(* PLC project Unnamed, Unknown Unnamed 1 *)
(* stored: creationDateTime 2024-09-03T16:04:08, modificationDateTime 2024-09-10T11:48:46 *)

PROGRAM irrigation_LD
  VAR
    SoilMoisture AT %IW0.0 : INT;  (* Soil moisture input from Modbus *)
  END_VAR
  VAR
    SoilMoistureMaxValue0 : INT := 500;  (* Soil moisture upper bound *)
  END_VAR
  VAR
    Temperature AT %IW0.1 : INT;  (* Temperature input from Modbus *)
    Humidity AT %IW0.2 : INT;  (* Humidity input from Modbus *)
    WaterFlow AT %IW0.3 : INT;  (* Water flow input from Modbus *)
    Pressure AT %QX0.4 : INT;  (* Pressure input from Modbus *)
    PumpControl AT %QX0.0 : BOOL;  (* Output to control the pump *)
    ValveControl AT %QX0.1 : BOOL;  (* Output to control the valve *)
  END_VAR
  VAR  (* added by the conversion: wires and edge detectors of the diagram *)
    _LE8_OUT : BOOL;
  END_VAR

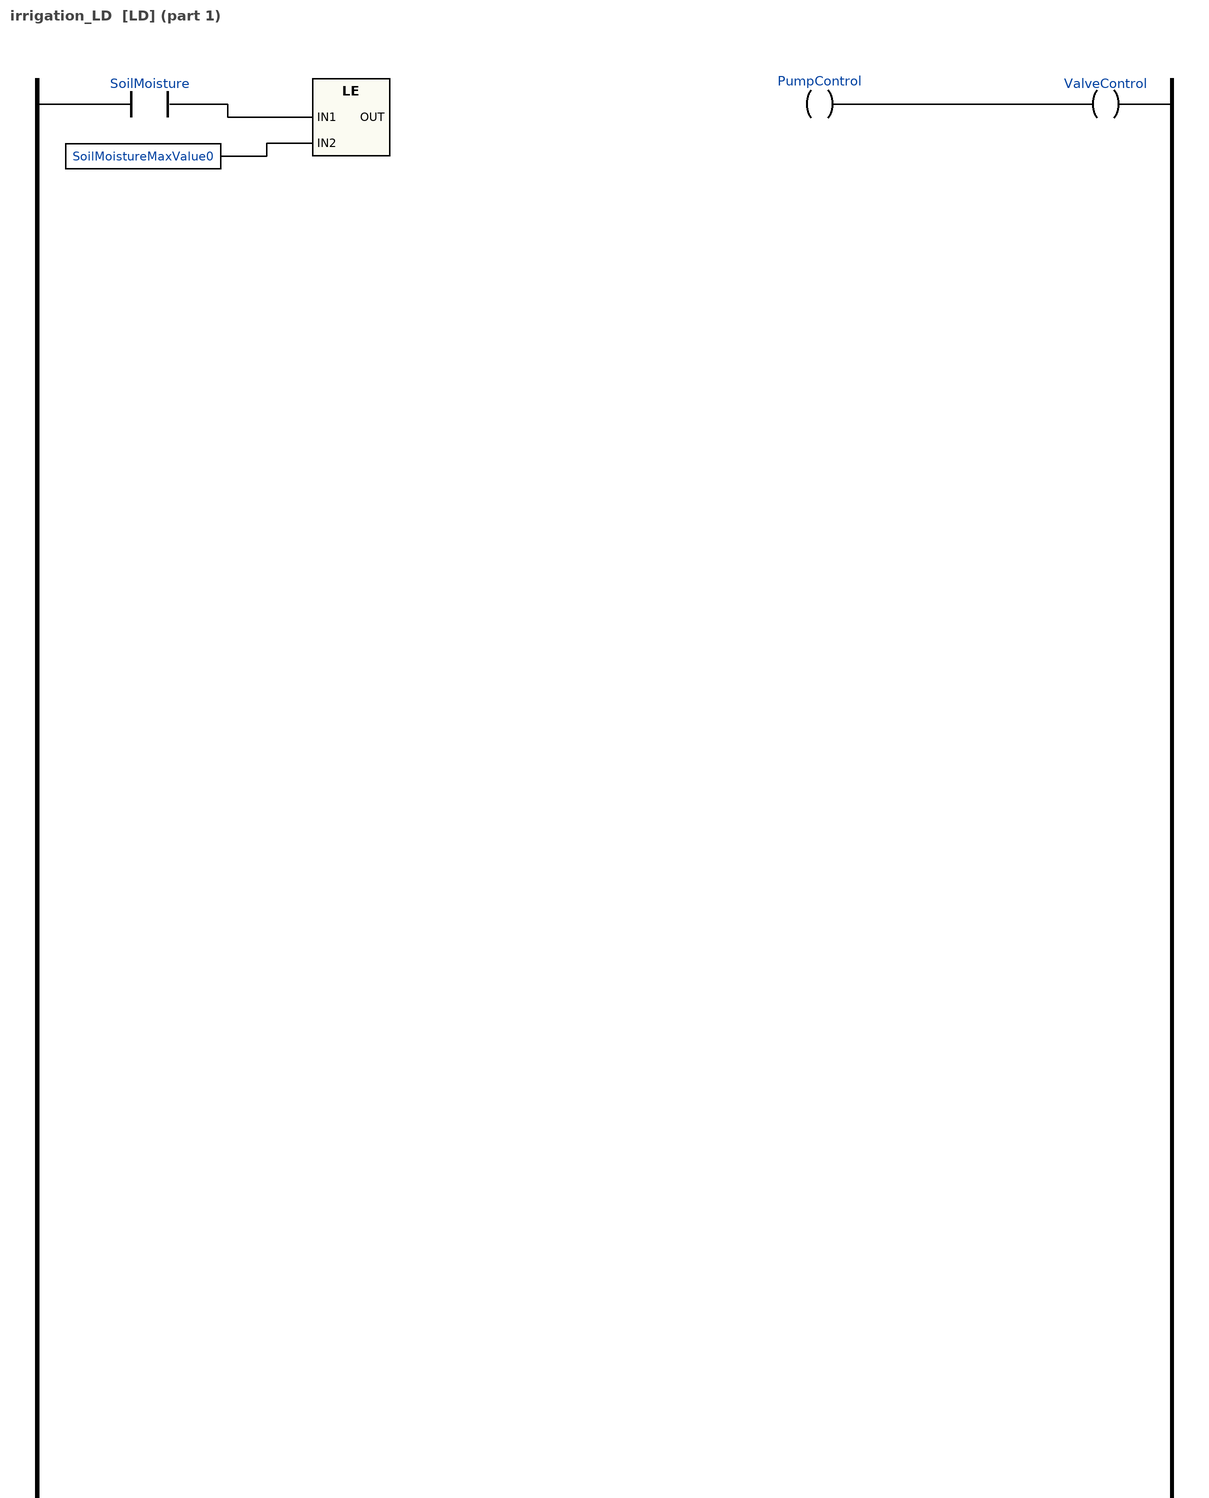
(* LD diagram, written out as Structured Text *)
_LE8_OUT := SoilMoisture <= SoilMoistureMaxValue0;
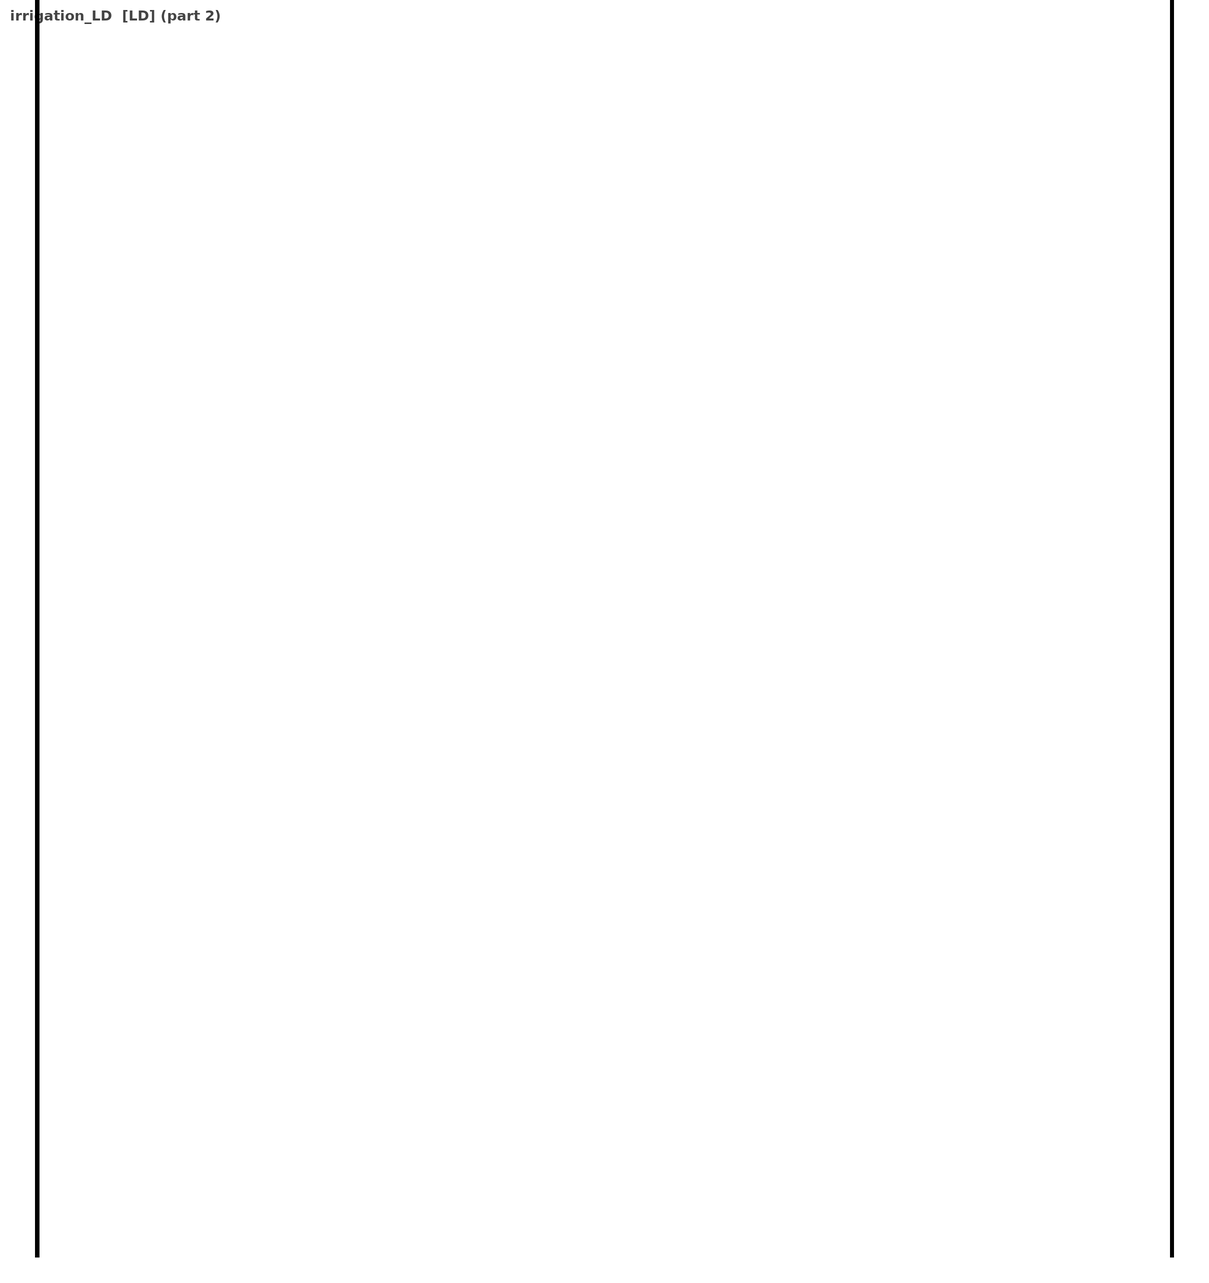
END_PROGRAM

PROGRAM irrigation_ST
  VAR
    SoilMoisture AT %IW0.0 : INT;  (* Soil moisture input from Modbus *)
    Temperature AT %IW0.1 : INT;  (* Temperature input from Modbus *)
    Humidity AT %IW0.2 : INT;  (* Humidity input from Modbus *)
    WaterFlow AT %IW0.3 : INT;  (* Water flow input from Modbus *)
    Pressure AT %QX0.4 : INT;  (* Pressure input from Modbus *)
    PumpControl AT %QX0.0 : BOOL;  (* Output to control the pump *)
    ValveControl AT %QX0.1 : BOOL;  (* Output to control the valve *)
  END_VAR

            // Structured Text code to control irrigation system

// Set the threshold values
VAR
    SoilMoistureThreshold : INT := 500;  // Moisture threshold for irrigation
    TempMin : INT := 20;                 // Minimum acceptable temperature
    TempMax : INT := 35;                 // Maximum acceptable temperature
    PressureMin : INT := 60;             // Minimum acceptable pressure
    PressureMax : INT := 140;            // Maximum acceptable pressure
    FlowMin : INT := 600;                // Minimum acceptable water flow
    FlowMax : INT := 950;                // Maximum acceptable water flow
END_VAR

// Main control logic
IF (SoilMoisture < SoilMoistureThreshold) THEN
    IF (Temperature > TempMin) AND (Temperature < TempMax) THEN
        IF (Pressure > PressureMin) AND (Pressure < PressureMax) THEN
            IF (WaterFlow > FlowMin) AND (WaterFlow < FlowMax) THEN
                // All conditions met, turn on the pump and open the valve
                PumpControl := TRUE;
                ValveControl := TRUE;
            ELSE
                // Water flow not in range, turn off the pump and valve
                PumpControl := FALSE;
                ValveControl := FALSE;
            END_IF;
        ELSE
            // Pressure not in range, turn off the pump and valve
            PumpControl := FALSE;
            ValveControl := FALSE;
        END_IF;
    ELSE
        // Temperature not in range, turn off the pump and valve
        PumpControl := FALSE;
        ValveControl := FALSE;
    END_IF;
ELSE
    // Soil moisture is sufficient, turn off the pump and valve
    PumpControl := FALSE;
    ValveControl := FALSE;
END_IF;

          
END_PROGRAM

CONFIGURATION Config0
  RESOURCE Res0 ON PLC
    TASK task0(INTERVAL := T#20ms, PRIORITY := 0);
    PROGRAM instance0 WITH task0 : irrigation_LD;
  END_RESOURCE
END_CONFIGURATION
